FUNCTION_BLOCK FB_EMbase
VAR
	TagName : STRING;
	Description : STRING;
	TagID : INT;
END_VAR

END_FUNCTION_BLOCK

(* stored: Version 1.1.0.1, ProductVersion 3.1.4024.12
   POU FB_EMbase: Id {d92c3cff-1ed3-441d-a6d7-7a26372df424}, SpecialFunc None *)
